// Standard CONCAT may return STRING(255). Explicit bounded copying preserves
// larger feedback objects and always leaves a terminating NUL in PLC memory.
used := LongStringLength(
    pText := ADR(destination),
    maxLength := 4095
);

count := LEN(fragment);
AppendDiagnosticText := used + count <= 4095;
IF NOT AppendDiagnosticText THEN RETURN; END_IF
outputBytes := ADR(destination);
inputBytes := ADR(fragment);
FOR i := 0 TO count - 1 DO outputBytes[used + i] := inputBytes[i]; END_FOR
outputBytes[used + count] := 0;

END_FUNCTION

// PLC/Application/LongStringLength
FUNCTION LongStringLength : INT
VAR_INPUT
    pText : POINTER TO BYTE;
    maxLength : INT;
END_VAR
VAR
    i : INT;
END_VAR

i := 0;
WHILE (i < maxLength) AND (pText[i] <> 0) DO
    i := i + 1;
END_WHILE;
LongStringLength := i;

END_FUNCTION

// PLC/Application/BuildDiagnosticFeedback
FUNCTION BuildDiagnosticFeedback : STRING(4095)
VAR
    output : STRING(4095);
    fragment : STRING(255);
    field : INT;
    i : INT;
    valid : BOOL;
    ok : BOOL := TRUE;
END_VAR

output := '{"currentPositions":[';
ok := TRUE;
FOR i := 1 TO 6 DO
    IF i > 1 THEN ok := AppendDiagnosticText(',', output) AND ok; END_IF
    ok := AppendDiagnosticText(REAL_TO_STRING(GVL.currentPositions[i].Number), output) AND ok;
END_FOR
ok := AppendDiagnosticText('],"diagnostics":{"version":1,"sequence":', output) AND ok;
DriveDiagnostics.sampleSequence := DriveDiagnostics.sampleSequence + 1;
ok := AppendDiagnosticText(UDINT_TO_STRING(DriveDiagnostics.sampleSequence), output) AND ok;
ok := AppendDiagnosticText(',"plcTickMs":', output) AND ok;
ok := AppendDiagnosticText(UDINT_TO_STRING(DriveDiagnostics.sampleTick), output) AND ok;
ok := AppendDiagnosticText(',"sdoReadErrors":', output) AND ok;
ok := AppendDiagnosticText(UDINT_TO_STRING(DriveDiagnostics.readErrorCount), output) AND ok;
ok := AppendDiagnosticText(',"positionUnit":"Festo user unit","velocityUnit":"Festo user unit/s","registerUnit":"raw CiA402","followingErrorSource":"0x60F4 readback","targetSource":"0x607A readback"', output) AND ok;
// Field order is fixed; actuator order stays A1..A6. Null means no new valid
// sample. SDO sample ticks are kept separately from packet assembly time.
FOR field := 1 TO 11 DO
    CASE field OF
        1: fragment := ',"receivedPositions":[';
        2: fragment := ',"receivedSpeeds":[';
        3: fragment := ',"actualPositions":[';
        4: fragment := ',"actualVelocities":[';
        5: fragment := ',"driveTargetPositions":[';
        6: fragment := ',"followingErrors":[';
        7: fragment := ',"targetSampleTickMs":[';
        8: fragment := ',"followingSampleTickMs":[';
        9: fragment := ',"sdoErrorIds":[';
        10: fragment := ',"requestedPositions":[';
        11: fragment := ',"requestedSpeeds":[';
    END_CASE
    ok := AppendDiagnosticText(fragment, output) AND ok;
    FOR i := 1 TO 6 DO
        IF i > 1 THEN ok := AppendDiagnosticText(',', output) AND ok; END_IF
        valid := TRUE;
        CASE field OF
            1: fragment := REAL_TO_STRING(TcpClient.servoData.positions[i].Number);
            2: fragment := REAL_TO_STRING(TcpClient.servoData.speeds[i].Number);
            3: fragment := REAL_TO_STRING(DriveDiagnostics.actualPositions[i]); valid := DriveDiagnostics.positionValid[i];
            4: fragment := REAL_TO_STRING(DriveDiagnostics.actualVelocities[i]); valid := DriveDiagnostics.velocityValid[i];
            5: fragment := LREAL_TO_STRING(DriveDiagnostics.driveTargets[i]); valid := DriveDiagnostics.targetNew[i];
            6: fragment := LREAL_TO_STRING(DriveDiagnostics.followingErrors[i]); valid := DriveDiagnostics.followingNew[i];
            7: fragment := UDINT_TO_STRING(DriveDiagnostics.targetTick[i]); valid := DriveDiagnostics.targetNew[i];
            8: fragment := UDINT_TO_STRING(DriveDiagnostics.followingTick[i]); valid := DriveDiagnostics.followingNew[i];
            9: fragment := UINT_TO_STRING(WORD_TO_UINT(DriveDiagnostics.readErrors[i]));
            10: fragment := REAL_TO_STRING(GVL.servoPositions[i]);
            11: fragment := REAL_TO_STRING(GVL.servoVelocities[i]);
        END_CASE
        IF NOT valid THEN fragment := 'null'; END_IF
        ok := AppendDiagnosticText(fragment, output) AND ok;
    END_FOR
    ok := AppendDiagnosticText(']', output) AND ok;
END_FOR
ok := AppendDiagnosticText('}}$N', output) AND ok;
IF ok THEN
    BuildDiagnosticFeedback := output;
    FOR i := 1 TO 6 DO
        DriveDiagnostics.targetNew[i] := FALSE;
        DriveDiagnostics.followingNew[i] := FALSE;
    END_FOR
ELSE
    // Never send truncated JSON. TcpClient counts this failure for inspection.
    BuildDiagnosticFeedback := '';
END_IF

END_FUNCTION

// PLC/Application/CSP_Receive
FUNCTION_BLOCK CSP_Receive
VAR_INPUT
    Connected : BOOL;
    Connection : CAA.HANDLE;
END_VAR
VAR_OUTPUT
    RejectedFrames, AcceptedFrames : UDINT;
    Error : BOOL;
END_VAR
VAR
    reader : NBS.TCP_Read;
    buffer : ARRAY[0..510] OF BYTE;
    count : UDINT;
    frame : STRING(511);
    length, i : INT;
    discarding : BOOL;
    positions : ARRAY[1..6] OF LREAL;
END_VAR

CSP_Data.Connected := Connected;
Error := FALSE;
IF NOT Connected THEN
    reader(xEnable:=FALSE); length := 0; discarding := FALSE; frame := ''; RETURN;
END_IF
reader(xEnable:=TRUE,hConnection:=Connection,szSize:=SIZEOF(buffer),pData:=ADR(buffer),szCount=>count);
IF reader.xReady AND count > 0 THEN
    FOR i := 0 TO UDINT_TO_INT(count)-1 DO
        IF buffer[i] = 10 THEN
            frame[length] := 0;
            IF NOT discarding AND length <= 254 AND CSP_ParseFrame(Frame:=frame,Positions:=positions) THEN
                CSP_Data.Generation := CSP_Data.Generation+1;
                CSP_Data.ReceivedPosition := positions; CSP_Data.ReceivedMode := 8;
                CSP_Data.ReceivedTick := TIME_TO_UDINT(TIME());
                CSP_Data.Generation := CSP_Data.Generation+1;
                AcceptedFrames := AcceptedFrames+1;
            ELSE RejectedFrames := RejectedFrames+1;
            END_IF
            length := 0; discarding := FALSE;
        ELSIF NOT discarding THEN
            IF length < 510 THEN frame[length] := buffer[i]; length := length+1;
            ELSE discarding := TRUE;
            END_IF
        END_IF
    END_FOR
END_IF
IF reader.xError THEN CSP_Data.Connected := FALSE; Error := TRUE; END_IF

END_FUNCTION_BLOCK

// PLC/Application/CSP_ParseFrame
FUNCTION CSP_ParseFrame : BOOL
VAR_INPUT
    Frame : STRING(511);
END_VAR
VAR_IN_OUT
    Positions : ARRAY[1..6] OF LREAL;
END_VAR
VAR
    parsed : ARRAY[1..6] OF LREAL;
    cursor, i : INT;
    speed : LREAL;
    prefix : STRING := '{"controlMode":8,"positions":[';
    middle : STRING := ',"speeds":[';
END_VAR

// Deliberately accept the exact compact schema emitted by BuildCommandPayload.
// Unknown fields/modes, missing/extra axes and legacy PP packets cannot move CSP.
CSP_ParseFrame := FALSE;
IF LEFT(Frame,LEN(prefix)) <> prefix THEN RETURN; END_IF
cursor := LEN(prefix);
FOR i := 1 TO 6 DO
    IF NOT CSP_ReadNumber(Text:=Frame,Cursor:=cursor,Number:=parsed[i]) THEN RETURN; END_IF
    IF i < 6 THEN
        IF Frame[cursor] <> 44 THEN RETURN; END_IF
    ELSE IF Frame[cursor] <> 93 THEN RETURN; END_IF
    END_IF
    cursor := cursor+1;
END_FOR
IF MID(Frame,LEN(middle),cursor+1) <> middle THEN RETURN; END_IF
cursor := cursor+LEN(middle);
FOR i := 1 TO 6 DO
    IF NOT CSP_ReadNumber(Text:=Frame,Cursor:=cursor,Number:=speed) OR speed <> 0 THEN RETURN; END_IF
    IF i < 6 THEN
        IF Frame[cursor] <> 44 THEN RETURN; END_IF
    ELSE IF Frame[cursor] <> 93 THEN RETURN; END_IF
    END_IF
    cursor := cursor+1;
END_FOR
IF Frame[cursor] <> 125 OR cursor+1 <> LEN(Frame) THEN RETURN; END_IF
Positions := parsed; CSP_ParseFrame := TRUE;

END_FUNCTION

// PLC/Application/CSP_ReadNumber
FUNCTION CSP_ReadNumber : BOOL
VAR_INPUT
    Text : STRING(511);
END_VAR
VAR_IN_OUT
    Cursor : INT;
    Number : LREAL;
END_VAR
VAR
    first, digits : INT;
    token : STRING(48);
END_VAR

// JSON number grammar, bounded token length. Reject malformed numbers instead
// of relying on STRING_TO_LREAL's permissive prefix conversion.
CSP_ReadNumber := FALSE; first := Cursor;
IF Text[Cursor] = 45 THEN Cursor := Cursor+1; END_IF
digits := 0;
IF Text[Cursor] = 48 THEN Cursor := Cursor+1; digits := 1;
ELSE
    WHILE Cursor <= LEN(Text) AND Text[Cursor] >= 48 AND Text[Cursor] <= 57 DO
        Cursor := Cursor+1; digits := digits+1;
    END_WHILE
END_IF
IF digits = 0 THEN RETURN; END_IF
IF Text[Cursor] = 46 THEN
    Cursor := Cursor+1; digits := 0;
    WHILE Cursor <= LEN(Text) AND Text[Cursor] >= 48 AND Text[Cursor] <= 57 DO
        Cursor := Cursor+1; digits := digits+1;
    END_WHILE
    IF digits = 0 THEN RETURN; END_IF
END_IF
IF Text[Cursor] = 101 OR Text[Cursor] = 69 THEN
    Cursor := Cursor+1;
    IF Text[Cursor] = 43 OR Text[Cursor] = 45 THEN Cursor := Cursor+1; END_IF
    digits := 0;
    WHILE Cursor <= LEN(Text) AND Text[Cursor] >= 48 AND Text[Cursor] <= 57 DO
        Cursor := Cursor+1; digits := digits+1;
    END_WHILE
    // C++ float exponents fit two digits. Bound before conversion so hostile
    // huge exponents cannot overflow the PLC's STRING_TO_LREAL conversion.
    IF digits = 0 OR digits > 2 THEN RETURN; END_IF
END_IF
IF Cursor-first > 48 THEN RETURN; END_IF
token := MID(Text, Cursor-first, first+1);
Number := STRING_TO_LREAL(token);
// All accepted numbers are finite and bounded; no NaN or Infinity refreshes watchdog.
CSP_ReadNumber := Number = Number AND ABS(Number) <= 1000000.0;

END_FUNCTION

// PLC/Application/CSP_Bezier
FUNCTION CSP_Bezier : LREAL
VAR_INPUT
    Points : ARRAY[0..5] OF LREAL;
    Degree : INT;
    U : LREAL;
END_VAR
VAR
    work : ARRAY[0..5] OF LREAL;
    i, k : INT;
END_VAR

// de Casteljau evaluation: bounded interpolation, including near endpoints.
work := Points;
FOR k := Degree TO 1 BY -1 DO
    FOR i := 0 TO k - 1 DO
        work[i] := (1.0 - U) * work[i] + U * work[i+1];
    END_FOR
END_FOR
CSP_Bezier := work[0];

END_FUNCTION

// PLC/Application/CSP_Brake
FUNCTION_BLOCK CSP_Brake
VAR_INPUT
    Start : BOOL;
    Position, Velocity, Acceleration : LREAL;
    StepSeconds, MaxAcceleration, MaxJerk : LREAL;
END_VAR
VAR_OUTPUT
    P, V, A, StopPosition : LREAL;
    Done, Valid : BOOL;
END_VAR
VAR
    t : ARRAY[1..3] OF LREAL;
    j : ARRAY[1..3] OF LREAL;
    phase : INT;
    sign, speed, accel, peak, h, remaining : LREAL;
    sp, sv, sa : LREAL;
    k : INT;
END_VAR

IF Start THEN
    P := Position; V := Velocity; A := Acceleration;
    Done := FALSE; Valid := FALSE; phase := 1;
    IF MaxJerk <= 0 OR MaxAcceleration <= 0 THEN RETURN; END_IF
    sign := 1.0;
    IF Velocity < 0 THEN sign := -1.0; END_IF
    speed := sign * Velocity; accel := sign * Acceleration;
    IF ABS(Velocity) < 1E-10 AND ABS(Acceleration) < 1E-10 THEN
        StopPosition := P; Done := TRUE; Valid := TRUE; RETURN;
    END_IF
    // Exact jerk-aware minimum stopping profile: -J, optional -A, +J.
    // A valid monotone trajectory must be able to unwind its braking acceleration
    // before velocity changes sign. Do not repair an invalid state by clamping V.
    IF accel < 0 AND speed + 1E-9 < accel * accel / (2.0 * MaxJerk) THEN RETURN; END_IF
    peak := MIN(MaxAcceleration, SQRT(MaxJerk * speed + accel * accel / 2.0));
    IF peak <= 0 THEN RETURN; END_IF
    t[1] := MAX(0.0, (accel + peak) / MaxJerk);
    t[2] := MAX(0.0, (speed + (accel*accel - 2.0*peak*peak)/(2.0*MaxJerk)) / peak);
    t[3] := peak / MaxJerk;
    j[1] := -sign * MaxJerk; j[2] := 0; j[3] := sign * MaxJerk;
    sp := P; sv := V; sa := A;
    FOR k := 1 TO 3 DO
        h := t[k];
        sp := sp + sv*h + sa*h*h/2.0 + j[k]*h*h*h/6.0;
        sv := sv + sa*h + j[k]*h*h/2.0;
        sa := sa + j[k]*h;
    END_FOR
    StopPosition := sp; Valid := TRUE;
    RETURN;
END_IF
IF Done OR NOT Valid THEN RETURN; END_IF
remaining := StepSeconds;
// Split a PLC interval at jerk-phase boundaries; never integrate beyond a stop.
FOR k := 1 TO 3 DO
    IF phase <= 3 THEN
        h := MIN(remaining, t[phase]);
        P := P + V*h + A*h*h/2.0 + j[phase]*h*h*h/6.0;
        V := V + A*h + j[phase]*h*h/2.0;
        A := A + j[phase]*h;
        t[phase] := t[phase] - h; remaining := remaining - h;
        IF t[phase] <= 1E-12 THEN phase := phase + 1; END_IF
    END_IF
END_FOR
IF phase > 3 THEN
    // Analytical terminal state, not a high-speed position clamp.
    P := StopPosition; V := 0; A := 0; Done := TRUE;
END_IF

END_FUNCTION_BLOCK

// PLC/Application/Main
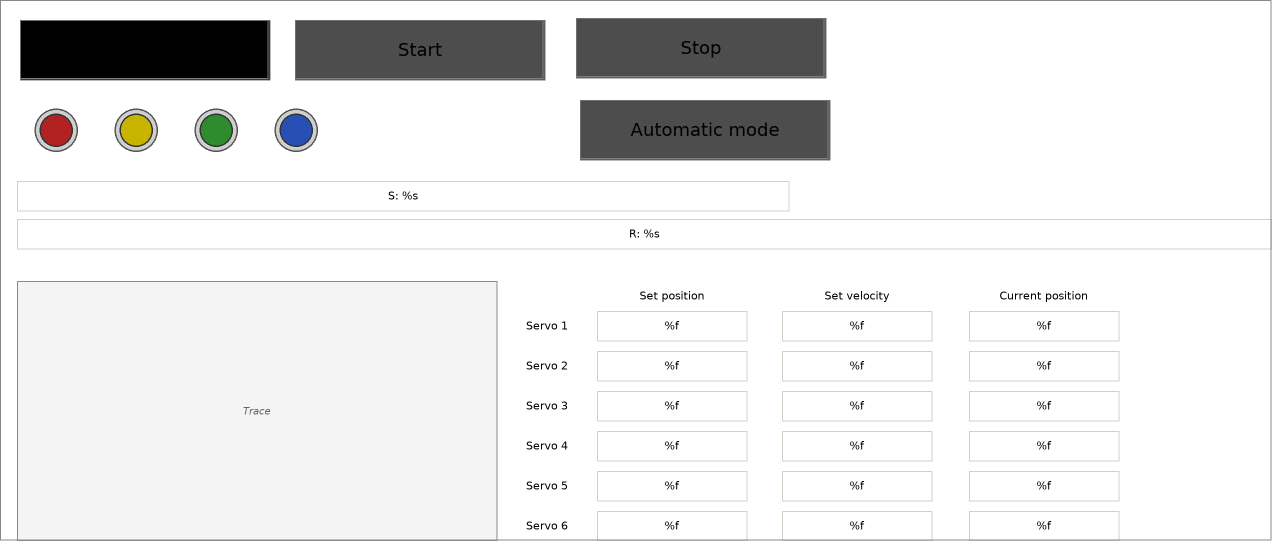
VISUALIZATION Main  // 1272x541
    Button (20,20 250x60), "Reset"
        tap GVL.resetHMI
    Button (295,20 250x60), "Start"
        tap GVL.startHMI
    Button (580,100 250x60), "Automatic mode"
        toggle GVL.usetcpdata
    Button (576,18 250x60), "Stop"
        tap GVL.stopHMI
    Lamp1 (191,105 50x50), variable: GVL.lightGreen, style: Lamp-Lamp1-Green
    Lamp1 (31,105 50x50), variable: GVL.lightRed, style: Lamp-Lamp1-Red
    Lamp1 (111,105 50x50), variable: GVL.lightYellow, style: Lamp-Lamp1-Yellow
    Textfield (17,181 772x30), "S: %s", text variable: TcpClient.sent
    Textfield (17,219 1255x30), "R: %s", text variable: TcpClient.received
    Textfield (597,311 150x30), "%f", text variable: GVL.servoPositions[1]
        OnMouseClick: write the text variable via InputWithLimits, min 0, max 400
    Textfield (597,351 150x30), "%f", text variable: GVL.servoPositions[2]
        OnMouseClick: write the text variable via InputWithLimits, min 0, max 400
    Textfield (597,391 150x30), "%f", text variable: GVL.servoPositions[3]
        OnMouseClick: write the text variable via InputWithLimits, min 0, max 400
    Textfield (597,431 150x30), "%f", text variable: GVL.servoPositions[4]
        OnMouseClick: write the text variable via InputWithLimits, min 0, max 400
    Textfield (597,471 150x30), "%f", text variable: GVL.servoPositions[5]
        OnMouseClick: write the text variable via InputWithLimits, min 0, max 400
    Textfield (597,511 150x30), "%f", text variable: GVL.servoPositions[6]
        OnMouseClick: write the text variable via InputWithLimits, min 0, max 400
    Textfield (782,311 150x30), "%f", text variable: GVL.servoVelocities[1]
        OnMouseClick: write the text variable via InputWithLimits, min 0, max 400
    Textfield (782,351 150x30), "%f", text variable: GVL.servoVelocities[2]
        OnMouseClick: write the text variable via InputWithLimits, min 0, max 400
    Textfield (782,391 150x30), "%f", text variable: GVL.servoVelocities[3]
        OnMouseClick: write the text variable via InputWithLimits, min 0, max 400
    Textfield (782,431 150x30), "%f", text variable: GVL.servoVelocities[4]
        OnMouseClick: write the text variable via InputWithLimits, min 0, max 400
    Textfield (782,471 150x30), "%f", text variable: GVL.servoVelocities[5]
        OnMouseClick: write the text variable via InputWithLimits, min 0, max 400
    Textfield (782,511 150x30), "%f", text variable: GVL.servoVelocities[6]
        OnMouseClick: write the text variable via InputWithLimits, min 0, max 400
    Label (597,281 150x30), "Set position"
    Label (782,281 150x30), "Set velocity"
    Label (497,311 100x30), "Servo 1"
    Label (497,351 100x30), "Servo 2"
    Label (497,391 100x30), "Servo 3"
    Label (497,431 100x30), "Servo 4"
    Label (497,471 100x30), "Servo 5"
    Label (497,511 100x30), "Servo 6"
    Lamp1 (271,105 50x50), variable: GVL.FlightSimulator.isReady(), style: Lamp-Lamp1-Blue
    Trace (17,281 480x260)
    Textfield (969,311 150x30), "%f", text variable: GVL.servoPositionsCurrent[1]
        OnMouseClick: write the text variable via InputWithLimits, min 0, max 400
    Textfield (969,351 150x30), "%f", text variable: GVL.servoPositionsCurrent[2]
        OnMouseClick: write the text variable via InputWithLimits, min 0, max 400
    Textfield (969,391 150x30), "%f", text variable: GVL.servoPositionsCurrent[3]
        OnMouseClick: write the text variable via InputWithLimits, min 0, max 400
    Textfield (969,431 150x30), "%f", text variable: GVL.servoPositionsCurrent[4]
        OnMouseClick: write the text variable via InputWithLimits, min 0, max 400
    Textfield (969,471 150x30), "%f", text variable: GVL.servoPositionsCurrent[5]
        OnMouseClick: write the text variable via InputWithLimits, min 0, max 400
    Textfield (969,511 150x30), "%f", text variable: GVL.servoPositionsCurrent[6]
        OnMouseClick: write the text variable via InputWithLimits, min 0, max 400
    Label (969,281 150x30), "Current position"
END_VISUALIZATION
